FUNCTION WRITE_PROTECTED_SINT
VAR_INPUT
    Ptr : POINTER TO SINT;
    Value : SINT;
END_VAR

Ptr^ := Value;

END_FUNCTION

(* stored: Version 1.1.0.1, ProductVersion 3.1.4022.18
   POU WRITE_PROTECTED_SINT: Id {e310eaa9-3123-4344-b07c-fc54b5c8e3ac}, SpecialFunc None *)
